INTERFACE I_BowlFeeder

PROPERTY Active : BOOL
GET
END_GET
END_PROPERTY

PROPERTY Busy : BOOL
GET
END_GET
END_PROPERTY

PROPERTY Error : BOOL
GET
END_GET
END_PROPERTY

METHOD MR_FirstCycle : BOOL
VAR_INPUT
	sName	: STRING;
END_VAR
END_METHOD

METHOD MR_Init : BOOL
VAR_INPUT
END_VAR
END_METHOD

METHOD MR_Start : BOOL
VAR_INPUT
END_VAR
END_METHOD

METHOD MR_Stop : BOOL
VAR_INPUT
END_VAR
END_METHOD

PROPERTY Running : BOOL
GET
END_GET
END_PROPERTY

PROPERTY Setpoint : REAL
GET
END_GET
SET
END_SET
END_PROPERTY

END_INTERFACE

(* stored: Version 1.1.0.1, ProductVersion 3.1.4024.9
   Itf I_BowlFeeder: Id {0ea241d8-ad4d-4c40-b136-02f1fa8cf02c}
   Property Active: Id {bd741382-8765-42d3-b030-a1b6e6e40f8b}
   Get Get: Id {4c99e76e-6751-4e6a-b0ff-66f00380cc2b}
   Property Busy: Id {cc424d09-e450-4306-bbcb-96eb2f0de43b}
   Get Get: Id {f6fdf655-3b44-485c-85e2-af1f9dbad275}
   Property Error: Id {14bd0ba7-24a0-40b4-997b-8555ae1b5dde}
   Get Get: Id {86194af5-983b-4467-8bde-1e385c13fe88}
   Method MR_FirstCycle: Id {5535c3a8-c7b9-421f-9860-715f1efd5974}
   Method MR_Init: Id {b88fc8cf-d8b8-466c-ab7e-d1c68b829a21}
   Method MR_Start: Id {a83232eb-4325-4d65-a524-0a08bacc05d7}
   Method MR_Stop: Id {02d75b9f-bb56-4ac4-b85b-ddbdaa40bdee}
   Property Running: Id {d503bc87-240b-4f23-9018-67d5f3ce0caa}
   Get Get: Id {3b8fd829-34f4-4074-84b8-27651eef013f}
   Property Setpoint: Id {7a55a89e-c787-4956-8266-91e9c325d0ac}
   Get Get: Id {6f301637-8992-4ade-a946-18592b09e4b5}
   Set Set: Id {f3188db2-4c0a-4644-af28-319ffca8b21d} *)
